Staubli VAL3: onF6Event.pgx

program onF6Event(bool& x_bSave[])
  local string l_sMessage
  local bool l_bYes
  local num l_nSize
  local num l_nFound
  local string l_sEvent
  local string l_sButton[2]
  local num l_nItem
begin
  // look if the bButton is enable
  if bButton[5]
    //
    // DELETE
    //
    call language:message(l_sMessage,80)
    call language:getYesNo(l_sButton)
    // ask the yes_no question
    call use:yes_no(l_sMessage,l_sButton,l_bYes)
    if l_bYes
      l_nItem=nIndexItem
      call trajType:getSizeItem(false,l_nSize)
      if l_nSize>1
        call trajType:deleteItem(nIndexItem)
        if nIndexItem>0
          nIndexItem=nIndexItem-1
        else
          nIndexItem=l_nItem
        endIf
        //refresh
        call buildList()
        use:bUseRefresh=true
      endIf
    endIf
    x_bSave=true
  endIf
end
